(*Usage:
 N.B. FILE BUFFER IS STORED IN THIS OBJECT, IN MEMORY.  DO NOT DO ACCESS ANOTHER FILE
 		WITH THIS BLOCK UNTIL YOU HAVE FINISHED WITH IT.
 		IF YOU WANT TO EXTEND THE LIFE OF THIS BUFFFER, CREATE A NEW ONE ELSEWHERE AND MEMCPY INTO IT!
 Call instance (i.e. FileRead();) every scan while waiting for operations to complete.
 SetFilePath()
 [OPTIONAL] StartCheckFileExists(); . Only recall if necessary (i.e. long time between file path set)
  
 StartRead();

 IF BufferAvailable
 use address and size indicated by DataBuffer and DataLength.
*)

FUNCTION_BLOCK INTERNAL T_FileReadBase
VAR
// backing properties
	_FilePath : Tc2_Utilities.T_MaxString;
	_Start : BOOL;
	_Busy : BOOL;
	_Done : BOOL;
	_Error : BOOL;
	_ErrorId : UDINT;
	_Read : BOOL; // if true, reads the file.
	_FileExists: BOOL; 
	_DataBuffer : POINTER TO BYTE; // remaining data (i.e. crc is stripped).
	_DataLength : UDINT;

// Function Block Objects
	FileOpen : FB_FileOpen; // Opens file 
	FileClose : FB_FileClose; // Closes file
	FileSeek : FB_FileSeek; // Move pointer to file position.
	FileTell	: FB_FileTell; // get file information.
	FileRead	: FB_FileRead; // read from file.
	
// Vars
	CheckFileExists : BOOL;		// when set true, check the file exists.
	FileHandle : UINT;			// file handle
	FileBufferSize : UDINT;			// size of file in bytes
	FileBuffer : POINTER TO BYTE; // holds file contents

// State Enum
	State : E_FileBaseStates := E_FileBaseStates.WaitForStart;
	
END_VAR

CASE State OF
	
	E_FileBaseStates.WaitForStart:	
		
		_Busy := FALSE;
		
		IF _Start THEN
			_Start := FALSE;
			_Busy := TRUE;
			_Done := FALSE;
			_Error := FALSE;
			_ErrorId := E_AdsErr.NOERR;
			FileHandle := 0;
			State := OpenFile;
			
			// delete pointer if it previously exists. 
			IF FileBuffer > 0 THEN 
				__DELETE(FileBuffer);
			END_IF
			
		END_IF

	E_FileBaseStates.OpenFile:
	
		FileOpen(bExecute := FALSE);
		
		FileOpen( 
			sNetId 		:= '', 
			sPathName 	:= _FilePath,
			nMode 		:= FOPEN_MODEREAD OR FOPEN_MODEBINARY, // Binary uses CRLF.
			bExecute 	:= TRUE);
		// Next Step
		State := WaitForOpenComplete;

	E_FileBaseStates.WaitForOpenComplete:
	
		FileOpen(bExecute	:= FALSE,
					hFile 		=> FileHandle,
					bError 		=> _Error,
					nErrId 		=> _ErrorId);
		
		IF NOT FileOpen.bBusy THEN
			_FileExists := NOT(_ErrorId = E_AdsErr.DEVICE_NOTFOUND); // check whether file exists.
			
			IF CheckFileExists THEN	
				// if checking whether a file exists, suppress error
				CheckFileExists := FALSE;
				_Error := FALSE;
				_ErrorId := 0;
				State := FinishAndCleanup;
				
			ELSE
				State := SEL(_Error, SeekEnd, FinishAndCleanup);
			END_IF
			
		END_IF

	E_FileBaseStates.SeekEnd:
	
		// move file pointer to end of file.
		FileSeek(bExecute := FALSE);
		
	 	FileSeek(
            sNetId		:= '', 
            hFile		:= FileHandle, 
            nSeekPos	:= 0, 
            eOrigin		:= E_SeekOrigin.SEEK_END, 
            bExecute	:= TRUE);
			
		State := WaitForSeekEndComplete;
			
	E_FileBaseStates.WaitForSeekEndComplete:
	
		FileSeek(bExecute	:= FALSE,
					bError 		=> _Error,
					nErrId 		=> _ErrorId);
		
		IF NOT FileSeek.bBusy THEN
			State := SEL(_Error, GetSize, FinishAndCleanup);
		END_IF
	
	E_FileBaseStates.GetSize:
	
		// As file pointer is at the end of the file, we can find size.
		FileTell(bExecute := FALSE);
		
		FileTell(
            sNetId		:= '', 
            hFile		:= FileHandle, 
            bExecute	:= TRUE, 
            tTimeout	:= );
		
		State := WaitForGetSizeComplete;
	
	E_FileBaseStates.WaitForGetSizeComplete:
	
		FileTell(bExecute 	:= FALSE,
					bError		=> _Error, 
					nErrId		=> _ErrorId, 
					nSeekPos	=> );
		
		IF NOT FileTell.bBusy THEN
			IF _Error THEN
				State :=  FinishAndCleanup;
			ELSE
				FileBufferSize := DINT_TO_UDINT(FileTell.nSeekPos);
				State := SeekStart;
			END_IF
	
		END_IF
	
	E_FileBaseStates.SeekStart:
	
		// move file pointer to end of file.
		FileSeek(bExecute := FALSE);
		
	 	FileSeek(
            sNetId		:= '', 
            hFile		:= FileHandle, 
            nSeekPos	:= 0, 
            eOrigin		:= E_SeekOrigin.SEEK_SET, 
            bExecute	:= TRUE);
			
		State := WaitForSeekStartComplete;
	
	E_FileBaseStates.WaitForSeekStartComplete:
	
		FileSeek(bExecute 	:= FALSE,
					bError 		=> _Error,
					nErrId 		=> _ErrorId);
		
		IF NOT FileSeek.bBusy THEN
			State := SEL(_Error, CreateBuffer, FinishAndCleanup);
		END_IF
	
	E_FileBaseStates.CreateBuffer:
	
		// create the buffer
		FileBuffer := __NEW(BYTE, FileBufferSize);
		
		IF FileBuffer > 0 THEN // if successfull
			State := ReadFromFile;
			
		ELSE // create buffer failed.
			_Error 	:= TRUE;
			_ErrorId 	:= 1802; // Out of memory
			State 		:= FinishAndCleanup;
			
		END_IF

	E_FileBaseStates.ReadFromFile:
	
		FileRead(bExecute := FALSE);
		
		FileRead(
            sNetId 		:= '', 
            hFile 		:= FileHandle, 
            pReadBuff 	:= FileBuffer, 
            cbReadLen 	:= FileBufferSize, 
            bExecute 	:= TRUE, 
            tTimeout 	:= );
			
		State := ReadFromFileComplete;
		
	E_FileBaseStates.ReadFromFileComplete:
	
		FileRead(bExecute := FALSE, 
					bError 		=> _Error, 
					nErrId 		=> _ErrorId);
		
		IF NOT FileRead.bBusy THEN
			State := SEL(_Error, CloseFile, FinishAndCleanup);
		END_IF
		
	E_FileBaseStates.CloseFile:	
	
		FileClose(bExecute := FALSE);
		
		FileClose(
			sNetId 		:= '',
			hFile 		:= FileHandle, 
			bExecute 	:= TRUE);
			
		// Next Step
		State := WaitForCloseComplete;

	E_FileBaseStates.WaitForCloseComplete:
	
		FileClose(bExecute := FALSE,
					bError 		=> _Error,
					nErrId 		=> _ErrorId);
					
		IF NOT FileClose.bBusy THEN
			FileHandle := 0;
			State := FinishAndCleanup;
		END_IF

	E_FileBaseStates.FinishAndCleanup: 
		
		_Done := TRUE;
		IF NOT _error THEN
			storeDataBufferAddressAndSizeIfValid();
		END_IF
		State := SEL(FileHandle <> 0, WaitForStart, CloseFile);
		
	ELSE // Error if we get here. Tidy up if we do.
		
		F_LogError(
			CONCAT('Illegal State request in FB_FileBase. Requested State: ', TO_STRING(State))
			);
		State := FinishAndCleanup; 

END_CASE

{attribute 'monitoring' := 'call'}
PROPERTY PUBLIC BufferAvailable : BOOL
GET
BufferAvailable := _DataBuffer > 0 AND_THEN _DataLength > 0;
END_GET
END_PROPERTY

{attribute 'monitoring' := 'call'}
PROPERTY PUBLIC Busy : BOOL
GET
Busy := _Busy;
END_GET
END_PROPERTY

{attribute 'monitoring' := 'call'}
PROPERTY PUBLIC DataBuffer : POINTER TO BYTE
GET
DataBuffer := _DataBuffer;
END_GET
END_PROPERTY

{attribute 'monitoring' := 'call'}
PROPERTY PUBLIC DataLength : UDINT
GET
DataLength := _DataLength;
END_GET
END_PROPERTY

{attribute 'monitoring' := 'call'}
PROPERTY PUBLIC Done : BOOL
GET
Done := _Done;
END_GET
END_PROPERTY

PROPERTY PUBLIC Error : BOOL
GET
Error := _Error;
END_GET
END_PROPERTY

{attribute 'monitoring' := 'call'}
PROPERTY PUBLIC ErrorId : UDINT
GET
ErrorId := _ErrorId;
END_GET
END_PROPERTY

METHOD FB_exit : BOOL
VAR_INPUT
	bInCopyCode : BOOL; // if TRUE, the exit method is called for exiting an instance that is copied afterwards (online change).
END_VAR
IF FileBuffer > 0 THEN
	__DELETE(FileBuffer);
END_IF
END_METHOD

{attribute 'monitoring' := 'call'}
PROPERTY PUBLIC FileExists : BOOL
GET
FileExists := _FileExists;
END_GET
END_PROPERTY

METHOD PUBLIC SetFilePath : BOOL
VAR_INPUT
	FilePath : Tc2_Utilities.T_MaxString;
END_VAR
IF State = WaitForStart THEN
	_FilePath := FilePath;
	SetFilePath := TRUE;
ELSE
	SetFilePath := FALSE;
END_IF
END_METHOD

METHOD PUBLIC StartCheckFileExists : BOOL
IF State = WaitForStart THEN
	CheckFileExists := TRUE;
	_Start := TRUE;
	StartCheckFileExists := TRUE;
ELSE
	StartCheckFileExists := FALSE;
END_IF
END_METHOD

METHOD PUBLIC StartRead : BOOL
//validate start is possible
IF State = WaitForStart THEN
	_Start := TRUE;
	_Read	:= TRUE;
END_IF

StartRead := _Start;
END_METHOD

METHOD PRIVATE storeDataBufferAddressAndSizeIfValid
_DataBuffer := FileBuffer;
_DataLength := FileBufferSize;
END_METHOD

END_FUNCTION_BLOCK

(* stored: Version 1.1.0.1, ProductVersion 3.1.4022.18
   POU T_FileReadBase: Id {0b68f5a6-75d9-48fc-a3e8-9282459b65be}, SpecialFunc None
   Folder Private: Id {a09af76c-4cc9-4509-a71e-1f4f13c838b2}
   Folder Properties: Id {aada1140-caa3-493b-8e3b-cf4165da8dc3}
   Property BufferAvailable: Id {98377ef3-a95a-4c75-b331-f39de9585bf8}
   Get Get: Id {30a1377a-211d-41dd-a7c4-98352e2d8f09}
   Property Busy: Id {57a1e3a6-2f68-46aa-b96f-df10bcc34601}
   Get Get: Id {74b775c8-9d8c-4ad4-815f-d94472e942e6}
   Property DataBuffer: Id {f6b2a83c-7a02-4aa6-b6a4-02f18458dbc0}
   Get Get: Id {0f2d0b3d-ff44-4397-bb77-7f2eea33e017}
   Property DataLength: Id {d036b2b9-ccc4-4aff-9b51-a6dccc677aae}
   Get Get: Id {9792ae36-ae30-4817-8617-61c55397b9b1}
   Property Done: Id {17a9325e-da93-4c8a-a8c0-86a326e86e72}
   Get Get: Id {4032a731-f3b1-4152-b5d0-762708aedfbb}
   Property Error: Id {75e8f711-3188-4cc3-8b9b-25083fa2b64c}
   Get Get: Id {eac10381-1173-4876-add8-d4707e2632d4}
   Property ErrorId: Id {d359406d-0387-4f26-9d01-1273710c3e19}
   Get Get: Id {8570eaf2-e7b8-440a-b37a-07ed61405b80}
   Method FB_exit: Id {fd4f5eea-e93e-4b5d-ab02-84bf37c9632f}
   Property FileExists: Id {727d6db5-f3eb-4edc-91a2-e76653e96821}
   Get Get: Id {c02442d1-a55b-44f6-953b-2b7372286d40}
   Method SetFilePath: Id {aa6478ba-4af4-49fd-845e-54cce517de49}
   Method StartCheckFileExists: Id {4f596f6e-1e68-447a-bbbd-e3b574a5eff2}
   Method StartRead: Id {3b23041b-2295-44d3-bb16-d270e002ae6c}
   Method storeDataBufferAddressAndSizeIfValid: Id {d5e7f845-e385-464f-baa8-ca80af23c95c} *)
